# EPICS StreamDevice protocol: group3hallprobeSup/group3hallprobe.proto
Terminator = CR LF;

init {
    out "A\$1 SE0GDR3GCNNUFG";
}

get_field {
    out "A\$1 F";
	in "%39c";
}

get_temp {
    out "A\$1 T";
	in "%f";
}

set_range {
    out "A\$1 R%d";
}
